FUNCTION_BLOCK FB_FlyPowerMarkManager
VAR_INPUT
	In : BOOL;
END_VAR
VAR_OUTPUT
	Out : BOOL;
END_VAR
VAR
	RTRIG_Enable	: R_TRIG;
	TON_DelayEnable	: TON;
END_VAR

TON_DelayEnable(IN := In, PT := T#1S);	
RTRIG_Enable(CLK := TON_DelayEnable.Q);

IF RTRIG_Enable.Q THEN
	Out := TRUE;
ELSIF NOT TON_DelayEnable.Q THEN
	Out := FALSE;
END_IF

END_FUNCTION_BLOCK

(* stored: Version 1.1.0.1, ProductVersion 3.1.4024.15
   POU FB_FlyPowerMarkManager: Id {26502597-14ae-42d2-8a73-1f4ca68823e0}, SpecialFunc None *)
